FUNCTION_BLOCK KeepCurrentOpCdtHMI (* Composite Function Block Type *)
  (* Standard: 61499-2 *)
  (* Version 0.0, 8/20/2024, SESA713705, Schneider Electric, template *)
  PACKAGE SE.Nereda;
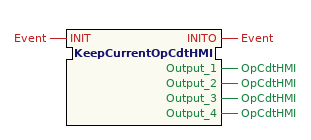
  EVENT_INPUT
    INIT;
  END_EVENT
  EVENT_OUTPUT
    INITO;
  END_EVENT
  PLUGS
    Output_1 : OpCdtHMI;
    Output_2 : OpCdtHMI;
    Output_3 : OpCdtHMI;
    Output_4 : OpCdtHMI;
  END_PLUGS
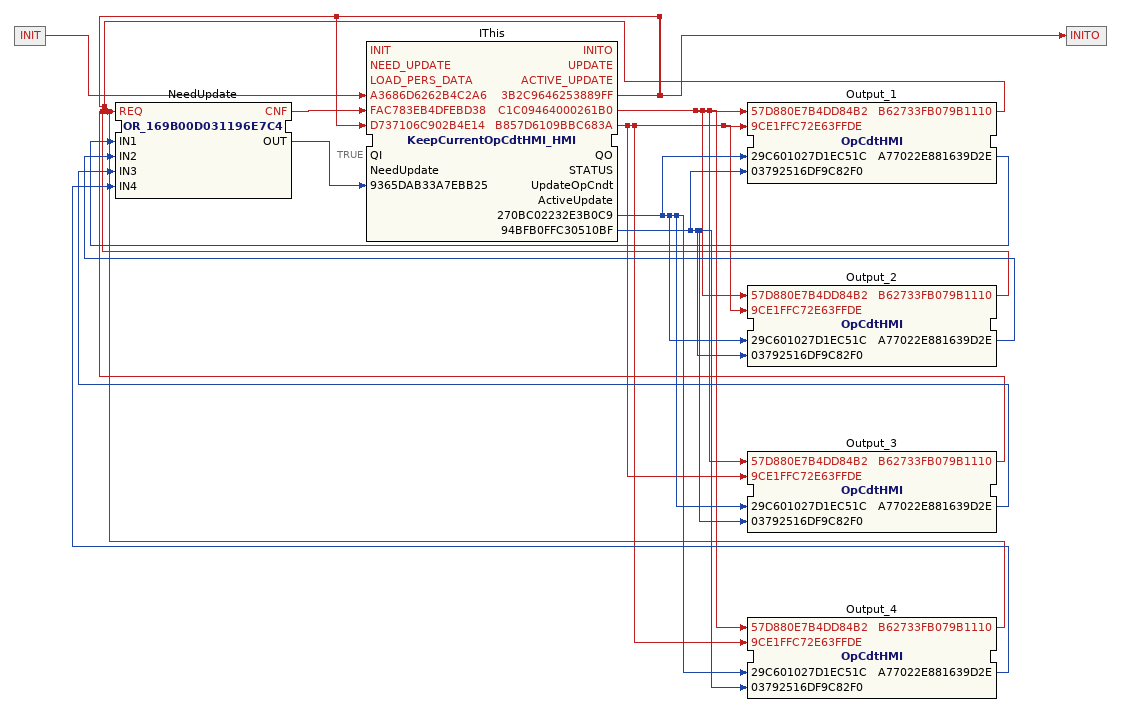
  FBS
    IThis : KeepCurrentOpCdtHMI_HMI(QI := TRUE);
    NeedUpdate : OR_169B00D031196E7C4; {SET_ATTRIBUTE(Configuration.GenericFBType.InterfaceParams, Runtime.Standard#CNT:=4;OUT:BOOL)}
  END_FBS
  EVENT_CONNECTIONS
    Output_1.B62733FB079B1110 TO NeedUpdate.REQ;
    Output_2.B62733FB079B1110 TO NeedUpdate.REQ;
    Output_3.B62733FB079B1110 TO NeedUpdate.REQ;
    Output_4.B62733FB079B1110 TO NeedUpdate.REQ;
    INIT TO IThis.A3686D6262B4C2A6;
    NeedUpdate.CNF TO IThis.FAC783EB4DFEBD38;
    IThis.3B2C9646253889FF TO IThis.D737106C902B4E14;
    IThis.3B2C9646253889FF TO INITO;
    IThis.3B2C9646253889FF TO NeedUpdate.REQ;
    IThis.C1C09464000261B0 TO Output_1.57D880E7B4DD84B2;
    IThis.C1C09464000261B0 TO Output_2.57D880E7B4DD84B2;
    IThis.C1C09464000261B0 TO Output_3.57D880E7B4DD84B2;
    IThis.C1C09464000261B0 TO Output_4.57D880E7B4DD84B2;
    IThis.B857D6109BBC683A TO Output_1.9CE1FFC72E63FFDE;
    IThis.B857D6109BBC683A TO Output_2.9CE1FFC72E63FFDE;
    IThis.B857D6109BBC683A TO Output_3.9CE1FFC72E63FFDE;
    IThis.B857D6109BBC683A TO Output_4.9CE1FFC72E63FFDE;
  END_CONNECTIONS
  DATA_CONNECTIONS
    Output_1.A77022E881639D2E TO NeedUpdate.IN1;
    Output_2.A77022E881639D2E TO NeedUpdate.IN2;
    NeedUpdate.OUT TO IThis.9365DAB33A7EBB25;
    IThis.270BC02232E3B0C9 TO Output_1.29C601027D1EC51C;
    IThis.270BC02232E3B0C9 TO Output_2.29C601027D1EC51C;
    IThis.270BC02232E3B0C9 TO Output_3.29C601027D1EC51C;
    IThis.270BC02232E3B0C9 TO Output_4.29C601027D1EC51C;
    IThis.94BFB0FFC30510BF TO Output_1.03792516DF9C82F0;
    IThis.94BFB0FFC30510BF TO Output_2.03792516DF9C82F0;
    IThis.94BFB0FFC30510BF TO Output_3.03792516DF9C82F0;
    IThis.94BFB0FFC30510BF TO Output_4.03792516DF9C82F0;
    Output_3.A77022E881639D2E TO NeedUpdate.IN3;
    Output_4.A77022E881639D2E TO NeedUpdate.IN4;
  END_CONNECTIONS
END_FUNCTION_BLOCK
